Staubli VAL3: HIT_YD.pjx

--- HIT_YD.pjx ---
Parameters version=s7.6.2 stackSize=5000 millimeterUnit=true
Program file=OMAC_Abort.pgx
Program file=OMAC_Hold.pgx
Program file=OMAC_Main.pgx
Program file=OMAC_Reset.pgx
Program file=OMAC_Start.pgx
Program file=OMAC_Stop.pgx
Program file=OMAC_Unhold.pgx
Program file=blow.pgx
Program file=bypassPick.pgx
Program file=cellManager.pgx
Program file=getToolStatus.pgx
Program file=goHome.pgx
Program file=init.pgx
Program file=initTracking.pgx
Program file=isInSafetyArea.pgx
Program file=modbusGet.pgx
Program file=modbusSet.pgx
Program file=overflowPick.pgx
Program file=Place.pgx
Program file=productionCycle.pgx
Program file=robot2PLC.pgx
Program file=send2NextRob.pgx
Program file=setAlarm.pgx
Program file=setConvSpeed.pgx
Program file=start.pgx
Program file=stop.pgx
Program file=trackErr_init.pgx
Program file=trackingPick.pgx
Program file=transferQueue.pgx
Data file=HIT_YD.dtx
Library alias=mot path=Disk://Tracking/Motion/Motion.pjx autoload=true password=
Type name=object path=Disk://Tracking/Templates/object/object.pjx

--- HIT_YD.dtx ---
aio aConvSpeed = {link=ModbusSrv-0\Modbus-Word\ao[3]}
aio aPlcCmd = {link=ModbusSrv-0\Modbus-Word\ai[0]}
aio aRbAlarm = {link=ModbusSrv-0\Modbus-Word\ao[0]}
aio aRbStatus = {link=ModbusSrv-0\Modbus-Word\ao[1]}
bool _bConvExist = true
bool _bEndCycle
bool _bIsPicking
bool _bIsPlacing
bool _bMutexCnvQueue = true
bool _bPartInTool
bool _bSentToHome = true
bool bLockPage
bool bPickDetection
bool bSetConvSpeed
bool bSyn
bool bTransferData
dio dAlarm[8]
  [0] = {link=ModbusSrv-0\Modbus-Bit\do[8]}
  [1] = {link=ModbusSrv-0\Modbus-Bit\do[9]}
  [2] = {link=ModbusSrv-0\Modbus-Bit\do[10]}
  [3] = {link=ModbusSrv-0\Modbus-Bit\do[11]}
  [4] = {link=ModbusSrv-0\Modbus-Bit\do[12]}
  [5] = {link=ModbusSrv-0\Modbus-Bit\do[13]}
  [6] = {link=ModbusSrv-0\Modbus-Bit\do[14]}
  [7] = {link=ModbusSrv-0\Modbus-Bit\do[15]}
dio dBlow = {link=BasicIO-1\%Q5}
dio dPartInTool = {link=fIn0}
dio dPermitPlace[4]
  [0] = {link=BasicIO-1\%I3}
  [1] = {link=BasicIO-1\%I2}
  [2] = {link=BasicIO-1\%I1}
  [3] = {link=BasicIO-1\%I0}
dio dPlaceDone[4]
  [0] = {link=BasicIO-1\%Q11}
  [1] = {link=BasicIO-1\%Q10}
  [2] = {link=BasicIO-1\%Q9}
  [3] = {link=BasicIO-1\%Q8}
dio dStartControl[4]
  [0] = {link=ModbusSrv-0\Modbus-Bit\di[4]}
  [1] = {link=ModbusSrv-0\Modbus-Bit\di[5]}
  [2] = {link=ModbusSrv-0\Modbus-Bit\di[6]}
  [3] = {link=ModbusSrv-0\Modbus-Bit\di[7]}
dio dStartState[4]
  [0] = {link=ModbusSrv-0\Modbus-Bit\do[4]}
  [1] = {link=ModbusSrv-0\Modbus-Bit\do[5]}
  [2] = {link=ModbusSrv-0\Modbus-Bit\do[6]}
  [3] = {link=ModbusSrv-0\Modbus-Bit\do[7]}
dio dVacuum = {link=BasicIO-1\%Q4}
frame fConveyor = {x=690.465999, y=-334.533545, z=-72.519533, rx=0.736674, ry=-0.299775, rz=179.886741, fatherId=world[0]}
frame fDetection = {x=319.933347, y=-456.969728, z=-77.119399, rx=1.134288, ry=-0.307561, rz=179.705392, fatherId=world[0]}
jointRs jDropPart = {j1=-61.262813, j2=45.342289, j3=74.332986, j4=152.342331}
jointRs jHome = {j1=-61.262813, j2=45.342289, j3=74.332986, j4=152.342331}
jointRs jPark = {j1=-61.262813, j2=45.342289, j3=74.332986, j4=152.342331}
mdesc _mLoad = {accel=77.44, vel=88, decel=77.44, leave=40, reach=40}
mdesc mLoad = {accel=121, vel=110, decel=121, leave=40, reach=40}
mdesc mNomSpeed = {accel=144, vel=120, decel=144, leave=20, reach=20}
mdesc mPickDown = {accel=169, vel=130, decel=169, blend=off, leave=30, reach=30}
mdesc mPickup = {accel=144, vel=120, decel=144}
mdesc mPlaceDown = {accel=144, vel=120, decel=144, blend=off, leave=15, reach=15}
mdesc mPlaceUp = {accel=169, vel=130, decel=169, blend=cartesian, leave=20, reach=20}
mdesc mSlow = {accel=1, vel=10, decel=1, leave=10, reach=10}
mdesc mUnload = {accel=144, vel=120, decel=144, leave=40, reach=40}
num _nBlowDelay
num _nCntBypassed
num _nCntPartsDone[2]
  [0] = 72643
  [1] = 72642
num _nCntTransfered = 4
num _nConvSpd
num _nCycleTime[4]
  [0] = 1.546
  [1] = 0.54
  [2] = 11.161
num _nCycleTimeIndx = 3
num _nID = -1
num _nLastStateCMD
num _nOmacStat = 3
num _nPartID = 1
num _nPlaceCurItem[2]
num _nPullIndexTQ
num _nPushIndexTQ
num _nStateCMD
num _nTimer = 369.505
num _nTrackErr = 3107
num nBlowID = 0.2
num nBypass
num nLoadRatio[4]
  [0] = 1.05
  [1] = 0.95
  [2] = 0.8
  [3] = 0.8
num nNomConvSpeed = 100
num nPartHeight = 5
num nPickAppro = 60
num nPickOS_X
num nPickOS_Y
num nPlaceAppro = 60
public num nPlaceNum = 4
num nSafeMaxX = 850
num nSafeMaxY
num nSafeMinX
num nSafeMinY = -650
num nStopTime = 0.02
num nTestData[5]
  [0] = 8
  [1] = -49
  [2] = 57
  [3] = 1
  [4] = 22760
num nVacuumID = 0.2
num nWaitDist2Up4BP = -150
num nWaitDistToDown = 50
num nWaitDistToUp[1 3]
  [0,0] = -70
  [0,1] = 140
  [0,2] = 400
num nWaitDistX = -130
object _oTransferQueue[1 100]
  [0,0]
    num nID = -1
    num nLatchedValue
    trsf trTrsf
  [0,1]
    num nID = -1
    num nLatchedValue
    trsf trTrsf
  [0,2]
    num nID = -1
    num nLatchedValue
    trsf trTrsf
  [0,3]
    num nID = -1
    num nLatchedValue
    trsf trTrsf
  [0,4]
    num nID = -1
    num nLatchedValue
    trsf trTrsf
  [0,5]
    num nID = -1
    num nLatchedValue
    trsf trTrsf
  [0,6]
    num nID = -1
    num nLatchedValue
    trsf trTrsf
  [0,7]
    num nID = -1
    num nLatchedValue
    trsf trTrsf
  [0,8]
    num nID = -1
    num nLatchedValue
    trsf trTrsf
  [0,9]
    num nID = -1
    num nLatchedValue
    trsf trTrsf
  [0,10]
    num nID = -1
    num nLatchedValue
    trsf trTrsf
  [0,11]
    num nID = -1
    num nLatchedValue
    trsf trTrsf
  [0,12]
    num nID = -1
    num nLatchedValue
    trsf trTrsf
  [0,13]
    num nID = -1
    num nLatchedValue
    trsf trTrsf
  [0,14]
    num nID = -1
    num nLatchedValue
    trsf trTrsf
  [0,15]
    num nID = -1
    num nLatchedValue
    trsf trTrsf
  [0,16]
    num nID = -1
    num nLatchedValue
    trsf trTrsf
  [0,17]
    num nID = -1
    num nLatchedValue
    trsf trTrsf
  [0,18]
    num nID = -1
    num nLatchedValue
    trsf trTrsf
  [0,19]
    num nID = -1
    num nLatchedValue
    trsf trTrsf
  [0,20]
    num nID = -1
    num nLatchedValue
    trsf trTrsf
  [0,21]
    num nID = -1
    num nLatchedValue
    trsf trTrsf
  [0,22]
    num nID = -1
    num nLatchedValue
    trsf trTrsf
  [0,23]
    num nID = -1
    num nLatchedValue
    trsf trTrsf
  [0,24]
    num nID = -1
    num nLatchedValue
    trsf trTrsf
  [0,25]
    num nID = -1
    num nLatchedValue
    trsf trTrsf
  [0,26]
    num nID = -1
    num nLatchedValue
    trsf trTrsf
  [0,27]
    num nID = -1
    num nLatchedValue
    trsf trTrsf
  [0,28]
    num nID = -1
    num nLatchedValue
    trsf trTrsf
  [0,29]
    num nID = -1
    num nLatchedValue
    trsf trTrsf
  [0,30]
    num nID = -1
    num nLatchedValue
    trsf trTrsf
  [0,31]
    num nID = -1
    num nLatchedValue
    trsf trTrsf
  [0,32]
    num nID = -1
    num nLatchedValue
    trsf trTrsf
  [0,33]
    num nID = -1
    num nLatchedValue
    trsf trTrsf
  [0,34]
    num nID = -1
    num nLatchedValue
    trsf trTrsf
  [0,35]
    num nID = -1
    num nLatchedValue
    trsf trTrsf
  [0,36]
    num nID = -1
    num nLatchedValue
    trsf trTrsf
  [0,37]
    num nID = -1
    num nLatchedValue
    trsf trTrsf
  [0,38]
    num nID = -1
    num nLatchedValue
    trsf trTrsf
  [0,39]
    num nID = -1
    num nLatchedValue
    trsf trTrsf
  [0,40]
    num nID = -1
    num nLatchedValue
    trsf trTrsf
  [0,41]
    num nID = -1
    num nLatchedValue
    trsf trTrsf
  [0,42]
    num nID = -1
    num nLatchedValue
    trsf trTrsf
  [0,43]
    num nID = -1
    num nLatchedValue
    trsf trTrsf
  [0,44]
    num nID = -1
    num nLatchedValue
    trsf trTrsf
  [0,45]
    num nID = -1
    num nLatchedValue
    trsf trTrsf
  [0,46]
    num nID = -1
    num nLatchedValue
    trsf trTrsf
  [0,47]
    num nID = -1
    num nLatchedValue
    trsf trTrsf
  [0,48]
    num nID = -1
    num nLatchedValue
    trsf trTrsf
  [0,49]
    num nID = -1
    num nLatchedValue
    trsf trTrsf
  [0,50]
    num nID = -1
    num nLatchedValue
    trsf trTrsf
  [0,51]
    num nID = -1
    num nLatchedValue
    trsf trTrsf
  [0,52]
    num nID = -1
    num nLatchedValue
    trsf trTrsf
  [0,53]
    num nID = -1
    num nLatchedValue
    trsf trTrsf
  [0,54]
    num nID = -1
    num nLatchedValue
    trsf trTrsf
  [0,55]
    num nID = -1
    num nLatchedValue
    trsf trTrsf
  [0,56]
    num nID = -1
    num nLatchedValue
    trsf trTrsf
  [0,57]
    num nID = -1
    num nLatchedValue
    trsf trTrsf
  [0,58]
    num nID = -1
    num nLatchedValue
    trsf trTrsf
  [0,59]
    num nID = -1
    num nLatchedValue
    trsf trTrsf
  [0,60]
    num nID = -1
    num nLatchedValue
    trsf trTrsf
  [0,61]
    num nID = -1
    num nLatchedValue
    trsf trTrsf
  [0,62]
    num nID = -1
    num nLatchedValue
    trsf trTrsf
  [0,63]
    num nID = -1
    num nLatchedValue
    trsf trTrsf
  [0,64]
    num nID = -1
    num nLatchedValue
    trsf trTrsf
  [0,65]
    num nID = -1
    num nLatchedValue
    trsf trTrsf
  [0,66]
    num nID = -1
    num nLatchedValue
    trsf trTrsf
  [0,67]
    num nID = -1
    num nLatchedValue
    trsf trTrsf
  [0,68]
    num nID = -1
    num nLatchedValue
    trsf trTrsf
  [0,69]
    num nID = -1
    num nLatchedValue
    trsf trTrsf
  [0,70]
    num nID = -1
    num nLatchedValue
    trsf trTrsf
  [0,71]
    num nID = -1
    num nLatchedValue
    trsf trTrsf
  [0,72]
    num nID = -1
    num nLatchedValue
    trsf trTrsf
  [0,73]
    num nID = -1
    num nLatchedValue
    trsf trTrsf
  [0,74]
    num nID = -1
    num nLatchedValue
    trsf trTrsf
  [0,75]
    num nID = -1
    num nLatchedValue
    trsf trTrsf
  [0,76]
    num nID = -1
    num nLatchedValue
    trsf trTrsf
  [0,77]
    num nID = -1
    num nLatchedValue
    trsf trTrsf
  [0,78]
    num nID = -1
    num nLatchedValue
    trsf trTrsf
  [0,79]
    num nID = -1
    num nLatchedValue
    trsf trTrsf
  [0,80]
    num nID = -1
    num nLatchedValue
    trsf trTrsf
  [0,81]
    num nID = -1
    num nLatchedValue
    trsf trTrsf
  [0,82]
    num nID = -1
    num nLatchedValue
    trsf trTrsf
  [0,83]
    num nID = -1
    num nLatchedValue
    trsf trTrsf
  [0,84]
    num nID = -1
    num nLatchedValue
    trsf trTrsf
  [0,85]
    num nID = -1
    num nLatchedValue
    trsf trTrsf
  [0,86]
    num nID = -1
    num nLatchedValue
    trsf trTrsf
  [0,87]
    num nID = -1
    num nLatchedValue
    trsf trTrsf
  [0,88]
    num nID = -1
    num nLatchedValue
    trsf trTrsf
  [0,89]
    num nID = -1
    num nLatchedValue
    trsf trTrsf
  [0,90]
    num nID = -1
    num nLatchedValue
    trsf trTrsf
  [0,91]
    num nID = -1
    num nLatchedValue
    trsf trTrsf
  [0,92]
    num nID = -1
    num nLatchedValue
    trsf trTrsf
  [0,93]
    num nID = -1
    num nLatchedValue
    trsf trTrsf
  [0,94]
    num nID = -1
    num nLatchedValue
    trsf trTrsf
  [0,95]
    num nID = -1
    num nLatchedValue
    trsf trTrsf
  [0,96]
    num nID = -1
    num nLatchedValue
    trsf trTrsf
  [0,97]
    num nID = -1
    num nLatchedValue
    trsf trTrsf
  [0,98]
    num nID = -1
    num nLatchedValue
    trsf trTrsf
  [0,99]
    num nID = -1
    num nLatchedValue
    trsf trTrsf
pointRs pPick = {shoulder=righty, fatherId=fDetection[0]}
pointRs pPlace[4]
  [0] = {x=752.590073, y=-120.83, z=-69.15, rx=180, rz=95, shoulder=righty, fatherId=world[0]}
  [1] = {x=614.985623, y=-120.83, z=-69.15, rx=180, rz=95, shoulder=righty, fatherId=world[0]}
  [2] = {x=480.25, y=-120.83, z=-69.15, rx=180, rz=95, shoulder=righty, fatherId=world[0]}
  [3] = {x=342.02, y=-120.83, z=-69.15, rx=180, rz=94.999983, shoulder=righty, fatherId=world[0]}
sio skToRobot = {link=Socket\toRobot_sk1}
sio toRobot1 = {link=Socket\synClient2}
string _sCycleStatus = "Waiting for part to pick"
string sConveyorList = "cvIn"
string sString = "done"
tool tGripper = {z=75, rz=-128, fatherId=flange[0], ioLink=valve1}

--- modbusSet.pgx ---
program modbusSet(num x_nNum (dimensions=1))
begin
  //通信正常，系统运行
  if (x_nNum==1)
    dStartState[0]=true
    dStartState[1]=false
    dStartState[2]=true
    dStartState[3]=false
    //通信正常，系统停止
  elseIf (x_nNum==2)
    dStartState[0]=true
    dStartState[1]=false
    dStartState[2]=false
    dStartState[3]=true
    //通信正常，系统复位
  elseIf (x_nNum==3)
    dStartState[0]=true
    dStartState[1]=true
    dStartState[2]=false
    dStartState[3]=false
    //0 通信准备，系统停止
  else
    dStartState[0]=true
    dStartState[1]=false
    dStartState[2]=false
    dStartState[3]=true
  endIf
end

--- OMAC_Start.pgx ---
program OMAC_Start()
  local point l_pHere
begin

  //OMAC进程:Starting
  _nOmacStat=2
  logMsg("上位机手动操作：启动")
  // Task for cell manager
  if taskStatus("cellManager")>=0
    taskKill("cellManager")
  endIf
  wait(taskStatus("cellManager")<0)
  taskCreate "cellManager",100,cellManager()
  wait(taskStatus("cellManager")==1)

  delay(0)
end

--- OMAC_Stop.pgx ---
program OMAC_Stop()
  local joint l_jHere
  local string l_sToolStatus
begin

  //OMAC进程:Stopping
  _nOmacStat=8
  logMsg("上位机手动操作：停止")
  stopMove()
  resetMotion()
  //
  // Stop task

  taskKill("cellManager")
  taskKill("overflowPick")
  taskKill("productionCycle")
  taskKill("Reset")
  taskKill("Start")
  taskKill("Hold")
  taskKill("Unhold")
  taskKill("Preheat")
  taskKill("openPallet")
  taskKill("changeBox")
  taskKill("convStopCheck")
  taskKill("TransferQueue1")
  taskKill("robot2PLC")

  resetMotion()
  while !isPowered()
    enablePower()
    delay(1)
  endWhile
  //
  // Move up axis 3
  l_jHere=herej()
  l_jHere.j3=95
  movej(l_jHere,tGripper,mSlow)
  //
  // Drop the part on the tool
  if bPickDetection==true
    call getToolStatus(l_sToolStatus)
  endIf
  if l_sToolStatus=="PartInTool" or !bPickDetection
    movej(jDropPart,tGripper,mSlow)
    waitEndMove()
    dVacuum=false
  else
    dVacuum=false
  endIf
  //
  // Go to park position
  movej(jPark,tGripper,mSlow)
  waitEndMove()
  wait(taskStatus("Reset")==-1)
  wait(taskStatus("Start")==-1)
  wait(taskStatus("Hold")==-1)
  wait(taskStatus("Unhold")==-1)
  wait(taskStatus("Preheat")==-1)
  wait(taskStatus("openPallet")==-1)
  wait(taskStatus("changeBox")==-1)
  wait(taskStatus("convStopCheck")==-1)
  wait(taskStatus("cellManager")==-1)
  wait(taskStatus("TransferQueue1")==-1)
  wait(taskStatus("overflowPick")==-1)
  wait(taskStatus("productionCycle")==-1)

  if _bConvExist
    call mot:kill()
    _bConvExist=false
  endIf

  disablePower()
  wait(isPowered()==false)
  //OMAC进程:Stopped
  _nOmacStat=9

  delay(0)
end

--- OMAC_Unhold.pgx ---
program OMAC_Unhold()
  local joint l_jHere
begin
  //OMAC进程:UnHolding
  _nOmacStat=7
  logMsg("上位机手动操作：恢复")
  resetMotion()
  call trackErr_init()
  enablePower()
  l_jHere=herej()
  l_jHere.j3=jHome.j3
  movej(l_jHere,tGripper,mSlow)
  movej(jHome,tGripper,mSlow)
  _bSentToHome=true
  waitEndMove()
  if taskStatus("cellManager")>=0
    taskKill("cellManager")
  endIf
  wait(taskStatus("cellManager")<0)
  taskCreate "cellManager",100,cellManager()
  wait(taskStatus("cellManager")==1)

  delay(0)
end

--- overflowPick.pgx ---
program overflowPick()
  local num l_nConvNum
  local num l_nConvSpeed
  local num l_nConvSpeedOld
  local num l_nDistDown
  local num l_nDistUp
  local num l_nEncLatchVal
  local num l_nError
  local num l_nLimCrossPer
begin
  // This program removes all the objects from the conveyor’s queue
  //  that the robot is not going to work with. It removes the
  //  objects by overflow or by bypass.
  // The use of this program on a task allows to remove the
  //  unnecessary objects from the conveyor’s queue while the robot
  //  is working with a previous object.
  // If the variable bTransferData is set to true, the program will
  //  send the objects to the transfer queue before removing the
  //  objects from the conveyor’s queue.
  // If the variable bSetConvSpeed is set to true, the program will
  //  reduce/stop the conveyor to avoid that an object leaves the
  //  tracking window.
  //
  // Input parameters
  //  None            :
  //
  // Output parameters
  //  None            :
  //
  //----------------------------------------------------------------
  //
  l_nConvNum=0
  l_nConvSpeed=0
  l_nConvSpeedOld=0
  //
  do
    //
    // Takes control of the Pick conveyor queue
    setMutex(_bMutexCnvQueue[l_nConvNum])
    //
    // Remove objects by Bypass
    if nBypass[l_nConvNum]>0 and _nCntBypassed[l_nConvNum]==0
      call bypassPick()
    endIf
    //
    // Check if there is an object on the conveyor’s queue
    if _nID[l_nConvNum]==-1
      call mot:getNextID(l_nConvNum,_nID[l_nConvNum])
    endIf
    //
    // If there is an object on the conveyor’s queue: Remove the object from the conveyor’s
    //  queue if the object has passed the downstream limit (overflow) or, if the variable
    //  setConvSpeed is set to true, stop the conveyor before the object crosses the downstream limit.
    if _nID[l_nConvNum]!=-1
      // Recover next object transformation from the stack
      call mot:getObjectData(l_nConvNum,pPick.trsf,l_nError)
      call mot:getDistance(l_nConvNum,pPick,0,l_nDistUp,l_nDistDown,l_nError)
      // Reduce/stop the speed of the conveyor when the object is in between the two middle limits.
      //  The value of the speed is calculated as a percentage of the nominal speed. The percentage
      //  is proportional to the distance of the object to the middle limits, 100% when the object
      //  is at the first middle limit and 0% when the object is at the second middle limit.
      if bSetConvSpeed[l_nConvNum] and l_nDistDown<nWaitDistToDown[l_nConvNum]
        l_nLimCrossPer=max((nWaitDistToUp[l_nConvNum,2]-l_nDistUp)/(nWaitDistToUp[l_nConvNum,2]-nWaitDistToUp[l_nConvNum,1]),0)
        l_nConvSpeed=l_nLimCrossPer*nNomConvSpeed[l_nConvNum]
        if l_nConvSpeedOld!=l_nConvSpeed
          call setConvSpeed(l_nConvNum,sel(l_nDistUp>nWaitDistToUp[l_nConvNum,1],l_nConvSpeed,nNomConvSpeed[l_nConvNum]))
          l_nConvSpeedOld=l_nConvSpeed
        endIf
      else
        // Remove objects by Overflow
        if (l_nDistUp>nWaitDistToUp[l_nConvNum,1])
          //
          // Send object to the next robot
          if bTransferData[l_nConvNum]
            call mot:getObjectLatch(l_nConvNum,l_nEncLatchVal,l_nError)
            call send2NextRob(l_nConvNum,_nID[l_nConvNum],pPick.trsf,l_nEncLatchVal)
          endIf
          //
          // Remove object from conveyor's queue
          call mot:removePart(l_nConvNum)
          _nID[l_nConvNum]=-1
          pPick.trsf={0,0,0,0,0,0}
          //
          _nCntTransfered[l_nConvNum]=_nCntTransfered[l_nConvNum]+1
        endIf
      endIf
    else
      // No object available => full speed on the conveyor
      l_nConvSpeed=nNomConvSpeed[l_nConvNum]
      if bSetConvSpeed[l_nConvNum] and l_nConvSpeedOld!=l_nConvSpeed
        call setConvSpeed(l_nConvNum,l_nConvSpeed)
        l_nConvSpeedOld=l_nConvSpeed
      endIf
    endIf
    //
    // Release control of the Pick conveyor queue.
    _bMutexCnvQueue[l_nConvNum]=false
    //
    delay(0)
  until false
end

--- Place.pgx ---
program place()
  local bool l_bNoError
  local joint l_jAppro
  local num l_nConvNum
  local num l_nError
  local num l_nMoveID
  local num l_nTrackStatus
  local pointRs l_pAppro
  local pointRs l_pPlace
  local string l_sToolStatus
begin
  l_nConvNum=1
  link(l_pPlace,world)
  //che modify start
  if nPlaceNum>3
    nPlaceNum=0
  endIf
  _mLoad=mLoad
  _mLoad.vel=mLoad.vel*nLoadRatio[nPlaceNum]
  _mLoad.accel=mLoad.accel*nLoadRatio[nPlaceNum]*nLoadRatio[nPlaceNum]
  _mLoad.decel=mLoad.decel*nLoadRatio[nPlaceNum]*nLoadRatio[nPlaceNum]

  //dControlVacuum[nPlaceNum]=false
  l_pPlace=pPlace[nPlaceNum]
  //end
  // Place part
  l_pAppro=appro(l_pPlace,{0,0,-nPlaceAppro,0,0,0})
  l_bNoError=pointToJoint(tGripper,jHome,l_pAppro,l_jAppro)
  call mot:getTrackStatus(l_nTrackStatus)
  if l_nTrackStatus>0
    // Use trackOff if the robot is synchronized
    if l_bNoError
      call mot:trackOffJ(l_jAppro,tGripper,_mLoad,l_nMoveID,l_nError)
    else
      call mot:trackOff(l_pAppro,tGripper,_mLoad,l_nMoveID,l_nError)
    endIf
  else
    // Use movej if the robot is not synchronized
    if l_bNoError
      l_nMoveID=movej(l_jAppro,tGripper,_mLoad)
    else
      l_nMoveID=movej(l_pAppro,tGripper,_mLoad)
    endIf
  endIf
  // wait permit signal
  wait(dPermitPlace[nPlaceNum]==true)
  l_nMoveID=movel(l_pPlace,tGripper,mPlaceDown)
  //Blow
  wait(getMoveId()>l_nMoveID+nBlowID)
  _nBlowDelay=0.3
  waitEndMove()
  delay(nStopTime)
  l_nMoveID=movel(l_pAppro,tGripper,mPlaceUp)
  // check PartInTool if bPickDetection
  if bPickDetection
    //wait(getMoveId()>l_nMoveID-0.8)
    wait(getMoveId()>l_nMoveID+nBlowID-1.1)
    call getToolStatus(l_sToolStatus)
  else
    wait(getMoveId()>l_nMoveID+nBlowID-1.1)
    _bPartInTool=false
  endIf
  // send done signal
  //dPlaceDone[nPlaceNum]=true
  wait(getMoveId()>l_nMoveID+0.1)
  delay(0)
  //dPlaceDone[nPlaceNum]=false
  if l_sToolStatus=="PartInTool" or _bPartInTool==false
    // A part has been placed
    _nCntPartsDone[l_nConvNum]=_nCntPartsDone[l_nConvNum]+1
  endIf
  delay(0)
  //che modify start
  delay(0)
  dPlaceDone[nPlaceNum]=true
  wait(getMoveId()>l_nMoveID+0.4)
  if nPlaceNum==3
    //toRobot1="done"
  endIf
  if nPlaceNum==3 and bSyn
    do
      sString=toRobot1
    until (sString=="done")
  endIf
  nPlaceNum=nPlaceNum+1
  nTestData[4]=nTestData[4]+1
end

--- productionCycle.pgx ---
program productionCycle()
  local bool l_bPartDone
  local string l_sToolStatus
begin
  // This program is the main cycle. It pick on part from the input
  // conveyor and places it on an empty cavity on the output conveyor.
  //
  // Input parameters
  //  None            :
  //
  // Output parameters
  //  None            :
  //
  //----------------------------------------------------------------
  //
  // In order to improve cycle time, vacuum is always on, even while
  //  placing a part. To place a part, the blow is activated for a
  //  short period of time when the robot arrives to the place position.
  //
  // Main loop

  call getToolStatus(l_sToolStatus)
  if (!bPickDetection and _bPartInTool==true) or (bPickDetection and l_sToolStatus=="PartInTool")
    call place()
  endIf
  //---------------------------------------------------------------------//
  toRobot1="done"
  do
    //Takes control of the Pick conveyor queue.
    setMutex(_bMutexCnvQueue[0])
    do
      call trackingPick(l_bPartDone)
      delay(0)
    until l_bPartDone
    // Release control of the Pick conveyor queue.
    _bMutexCnvQueue[0]=false

    //
    call place()
    //
    delay(0)
  until _bEndCycle
  _bEndCycle=true
  //
end

--- setAlarm.pgx ---
program setAlarm(num x_nNum (dimensions=1))
begin
  if (x_nNum==0)
    dAlarm[0]=true
    dAlarm[1]=false
    dAlarm[2]=false
    dAlarm[3]=false
    dAlarm[4]=false
    dAlarm[5]=false
    dAlarm[6]=false
    dAlarm[7]=false
  elseIf (x_nNum==1)
    dAlarm[0]=false
    dAlarm[1]=true
    dAlarm[2]=false
    dAlarm[3]=false
    dAlarm[4]=false
    dAlarm[5]=false
    dAlarm[6]=false
    dAlarm[7]=false
  elseIf (x_nNum==2)
    dAlarm[0]=false
    dAlarm[1]=false
    dAlarm[2]=true
    dAlarm[3]=false
    dAlarm[4]=false
    dAlarm[5]=false
    dAlarm[6]=false
    dAlarm[7]=false
  elseIf (x_nNum==3)
    dAlarm[0]=false
    dAlarm[1]=false
    dAlarm[2]=true
    dAlarm[3]=false
    dAlarm[4]=false
    dAlarm[5]=false
    dAlarm[6]=false
    dAlarm[7]=false
  elseIf (x_nNum==4)
    dAlarm[0]=false
    dAlarm[1]=false
    dAlarm[2]=false
    dAlarm[3]=false
    dAlarm[4]=true
    dAlarm[5]=false
    dAlarm[6]=false
    dAlarm[7]=false
  elseIf (x_nNum==5)
    dAlarm[0]=false
    dAlarm[1]=false
    dAlarm[2]=false
    dAlarm[3]=false
    dAlarm[4]=false
    dAlarm[5]=true
    dAlarm[6]=false
    dAlarm[7]=false
  elseIf (x_nNum==6)
    dAlarm[0]=false
    dAlarm[1]=false
    dAlarm[2]=false
    dAlarm[3]=false
    dAlarm[4]=false
    dAlarm[5]=false
    dAlarm[6]=true
    dAlarm[7]=false
  elseIf (x_nNum==7)
    dAlarm[0]=false
    dAlarm[1]=false
    dAlarm[2]=false
    dAlarm[3]=false
    dAlarm[4]=false
    dAlarm[5]=false
    dAlarm[6]=false
    dAlarm[7]=true
  else
    dAlarm[0]=false
    dAlarm[1]=false
    dAlarm[2]=false
    dAlarm[3]=false
    dAlarm[4]=false
    dAlarm[5]=false
    dAlarm[6]=false
    dAlarm[7]=false

  endIf
end
